(* IEC 61131-3 sources: learning-path/04_introduction_to_st/exercises/3_extend_tank_functionality/src, 2 files *)

(* ---- valve.st ---- *)
NAMESPACE Siemens.AxTraining.ControlModules

    FUNCTION_BLOCK Valve
        VAR_INPUT
            cmdOpen :BOOL;
            cmdClose: BOOL;
        END_VAR
        VAR_OUTPUT
            ctrlOpen :BOOL;
            ctrlClose : BOOL;
        END_VAR

        ctrlClose := FALSE;
        ctrlOpen := FALSE;
        IF cmdClose THEN
            ctrlClose := TRUE;
        ELSIF cmdOpen THEN
            ctrlOpen := TRUE;
        END_IF;

    END_FUNCTION_BLOCK

END_NAMESPACE

(* ---- fluidProgram.st ---- *)
USING Siemens.AxTraining.EquipmentModules;

NAMESPACE Siemens.AxTraining
    PROGRAM FluidProgram

        VAR_EXTERNAL
            cmdFillTank : BOOL;
            cmdEmptyTank : BOOL;
            inletOpenTank : BOOL;
            outletOpenTank : BOOL;
        END_VAR
        VAR
            tank : Tank;
        END_VAR

        tank(cmdFill := cmdFillTank,
            cmdEmpty := cmdEmptyTank,
            inletOpen => inletOpenTank,
            outletOpen => outletOpenTank);
    END_PROGRAM
END_NAMESPACE
